// TIA Portal V16 export
// export: Created 2024-09-05T17:39:11.0923044Z, ExportSetting WithDefaults, DisplayName Totally Integrated Automation Portal, DisplayVersion V16 Update 6, DisplayName TIA Portal Version Control Interface, DisplayVersion V16 Update 2, DisplayName TIA Portal Openness, DisplayVersion V16 Update 6, DisplayName STEP 7 Professional, DisplayVersion V16 Update 6, DisplayName STEP 7 Safety, DisplayVersion V16, DisplayName WinCC Advanced, DisplayVersion V16 Update 6
DATA_BLOCK "Devices_Diagnostic_DB"   // DB8
VERSION : 0.1
// stored: AutoNumber true, DBAccessibleFromOPCUA true, InstanceOfName Devices_Diagnostic, InstanceOfType FB
"Devices_Diagnostic"
   // VAR_INPUT
   //    DPIdentifier : HW_IOSYSTEM := 301;
   //    PNIdentifier : HW_IOSYSTEM := 264;
   // END_VAR
   // VAR_OUTPUT
   //    PNmissing : Bool;
   // END_VAR
   // VAR
   //    PNConfigured : Array[0..1023] of Bool;
   //    PNFaulty : Array[0..1023] of Bool;
   //    PNDisabled : Array[0..1023] of Bool;
   //    PNExist : Array[0..1023] of Bool;
   //    DPConfigured : Array[0..1023] of Bool;
   //    DPFaulty : Array[0..1023] of Bool;
   //    DPDisabled : Array[0..1023] of Bool;
   //    DPExist : Array[0..1023] of Bool;
   // END_VAR
BEGIN
   PNConfigured[0] := TRUE;
   PNConfigured[1..10] := FALSE;
   PNConfigured[11] := TRUE;
   PNConfigured[12..30] := FALSE;
   PNConfigured[31..34] := TRUE;
   PNConfigured[35..40] := FALSE;
   PNConfigured[41] := TRUE;
   PNConfigured[42..60] := FALSE;
   PNConfigured[61..66] := TRUE;
   PNConfigured[67] := FALSE;
   PNConfigured[68..71] := TRUE;
   PNConfigured[72] := FALSE;
   PNConfigured[73..74] := TRUE;
   PNConfigured[75..90] := FALSE;
   PNConfigured[91] := TRUE;
   PNConfigured[92..1023] := FALSE;
   PNFaulty[0..1023] := FALSE;
   PNDisabled[0..1023] := FALSE;
   PNExist[0] := TRUE;
   PNExist[1..10] := FALSE;
   PNExist[11] := TRUE;
   PNExist[12..30] := FALSE;
   PNExist[31..34] := TRUE;
   PNExist[35..40] := FALSE;
   PNExist[41] := TRUE;
   PNExist[42..60] := FALSE;
   PNExist[61..66] := TRUE;
   PNExist[67] := FALSE;
   PNExist[68..71] := TRUE;
   PNExist[72] := FALSE;
   PNExist[73..74] := TRUE;
   PNExist[75..90] := FALSE;
   PNExist[91] := TRUE;
   PNExist[92..1023] := FALSE;
   DPConfigured[0..1023] := FALSE;
   DPFaulty[0..1023] := FALSE;
   DPDisabled[0..1023] := FALSE;
   DPExist[0..1023] := FALSE;
END_DATA_BLOCK
